Omron Sysmac Studio project ewon_iolink (Sysmac Studio 1.57.0.7, StandardProject)

# Controller new_Controller_0: NX1P2-1040DT1 version 1.18
Task PrimaryTask (priority 4, period or condition 2000): Programa0

TYPE u_byte_array_to_word : UNION
    input : ARRAY[0..1] OF BYTE;
    output : WORD;
END_UNION END_TYPE
TYPE t_nivel : STRUCT
    detectando : BOOL;
    distancia : INT;
END_STRUCT END_TYPE

VAR_GLOBAL
    s_nivel : ARRAY[0..1] OF BYTE;  (* at IOBus://unit#2/Port1 Input Data01 *)
    s_temperatura : ARRAY[0..1] OF BYTE;  (* at IOBus://unit#2/Port2 Input Data01 *)
END_VAR
VAR_GLOBAL RETAIN
    temperatura AT %D800 : REAL;
    sensor_capacitivo AT %D808 : t_nivel;
END_VAR

PROGRAM Programa0
VAR
    convertir_nivel : u_byte_array_to_word;
    convertir_temperatura : u_byte_array_to_word;
END_VAR
VAR_EXTERNAL
    s_nivel : ARRAY[0..1] OF BYTE;
    s_temperatura : ARRAY[0..1] OF BYTE;
    temperatura : REAL;
    sensor_capacitivo : t_nivel;
END_VAR

(* Section Sección0: ladder, written here as Structured Text *)

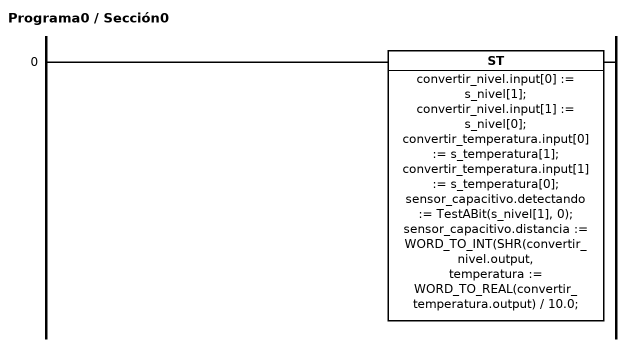
(* Rung 0 *)
convertir_nivel.input[0] := s_nivel[1];
convertir_nivel.input[1] := s_nivel[0];

convertir_temperatura.input[0] := s_temperatura[1];
convertir_temperatura.input[1] := s_temperatura[0];

sensor_capacitivo.detectando := TestABit(s_nivel[1], 0);
sensor_capacitivo.distancia := WORD_TO_INT(SHR(convertir_nivel.output, 1));

temperatura := WORD_TO_REAL(convertir_temperatura.output) / 10.0;
END_PROGRAM